# EPICS substitutions: modules/event/evrSupport/Db/ioc/IOC-IN20-BP01Testevr.substitutions
#==============================================================================
#
# Abs:  LCLS EVR IOC records for Test IN20 BP01
#
# Name: IOC-IN20-BP01Testevr.substitutions
#
#==============================================================================
#
file evrBPXX.db
{
pattern { DEV           }
	{ EVR:IN20:BP01 }
}
